SUBAPPLICATION Zaehler (* Subapplication Type *)
  (* Standard: 61499-2 *)
  (* Version 1.0, 2023-02-17, Franz *)
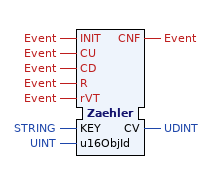
  EVENT_INPUT
    INIT; (* Initialization Request *)
    CU; (* Count Up *)
    CD; (* Count Down *)
    R; (* Reset *)
    rVT; (* refresh VT *)
  END_EVENT
  EVENT_OUTPUT
    CNF; (* Confirmation -- Counter Value was changed *)
  END_EVENT
  VAR_INPUT
    KEY : STRING;
    u16ObjId : UINT;
  END_VAR
  VAR_OUTPUT
    CV : UDINT; (* Counter Value *)
  END_VAR
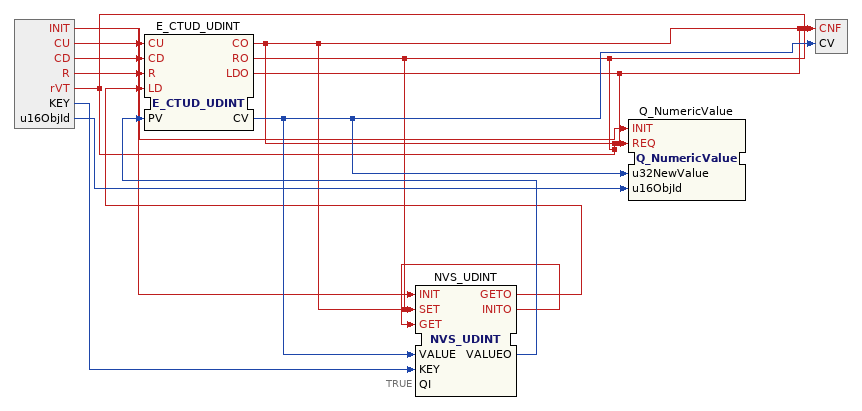
  FBS
    E_CTUD_UDINT : E_CTUD_UDINT;
    Q_NumericValue : Q_NumericValue;
    NVS_UDINT : NVS_UDINT(QI := TRUE);
  END_FBS
  EVENT_CONNECTIONS
    INIT TO Q_NumericValue.INIT;
    E_CTUD_UDINT.CO TO Q_NumericValue.REQ;
    E_CTUD_UDINT.RO TO Q_NumericValue.REQ;
    E_CTUD_UDINT.LDO TO Q_NumericValue.REQ;
    CU TO E_CTUD_UDINT.CU;
    CD TO E_CTUD_UDINT.CD;
    R TO E_CTUD_UDINT.R;
    INIT TO NVS_UDINT.INIT;
    E_CTUD_UDINT.CO TO NVS_UDINT.SET;
    E_CTUD_UDINT.RO TO NVS_UDINT.SET;
    NVS_UDINT.GETO TO E_CTUD_UDINT.LD;
    NVS_UDINT.INITO TO NVS_UDINT.GET;
    E_CTUD_UDINT.CO TO CNF;
    E_CTUD_UDINT.RO TO CNF;
    E_CTUD_UDINT.LDO TO CNF;
    rVT TO Q_NumericValue.REQ;
    rVT TO CNF;
  END_CONNECTIONS
  DATA_CONNECTIONS
    E_CTUD_UDINT.CV TO Q_NumericValue.u32NewValue;
    E_CTUD_UDINT.CV TO NVS_UDINT.VALUE;
    NVS_UDINT.VALUEO TO E_CTUD_UDINT.PV;
    E_CTUD_UDINT.CV TO CV;
    u16ObjId TO Q_NumericValue.u16ObjId;
    KEY TO NVS_UDINT.KEY;
  END_CONNECTIONS
END_SUBAPPLICATION
